FUNCTION GetTickCount : LINT
VAR_INPUT
END_VAR
VAR
	
END_VAR
VAR_STAT
	GST: Tc2_System.GETCPUCOUNTER;
END_VAR

GST();
GetTickCount := LWORD_TO_LINT(((DWORD_TO_LWORD(GST.cpuCntHiDW) * 16#100000000) + GST.cpuCntLoDW)) / 10000;

END_FUNCTION

(* stored: Version 1.1.0.1, ProductVersion 3.1.4024.6
   POU GetTickCount: Id {60465d36-94d5-4bba-aeb4-47818b21e733}, SpecialFunc None *)
